// TIA Portal V16 export
// export: Created 2021-07-12T14:47:20.993443Z, ExportSetting WithDefaults, DisplayName Totally Integrated Automation Portal, DisplayVersion V16, DisplayName TIA Portal Version Control Interface, DisplayVersion V16, DisplayName TIA Portal Openness, DisplayVersion V16, DisplayName STEP 7 Professional, DisplayVersion V16, DisplayName STEP 7 Safety, DisplayVersion V16, DisplayName WinCC Professional, DisplayVersion V16
TYPE "SimaHydTO_typeHMIConnectionVCharEditorTable"
TITLE = SimaHydTO_typeHMIConnectionVCharEditorTable
// HMI interface: VChar editor
// stored: IsFailsafeCompliant false
   STRUCT
      Appearance : Array[0..20] of Int;   // 0: invisible / 1: visible / 2: selected
      Index : Array[0..20] of Int;
      Velocity : Array[0..20] of Real;
      QOutput : Array[0..20] of Real;
      VelocityLimitPositive : Real;   // Max velocity in positive direction
      VelocityLimitNegative : Real;   // Max velocity in negative direction
      ZeroZonePositive : Real;   // Overlapping zone of valve in positive direction
      ZeroZoneNegative : Real;   // Overlapping zone of valve in negative direction
   END_STRUCT;
END_TYPE
